PROGRAM FB_Window
VAR
END_VAR
VAR_INPUT
	dataAxis: typeDataAxis;
	optionA:typeVectorOptions;
	optionB:typeVectorOptions;
//	optionC:typeVectorOptions;
//	optionD:typeVectorOptions;
END_VAR

(*
	
	^
	value
	|
	|							C
	|			1_______________________________4
	|			|								|
	|			|								|
	|			|								|
	|			|								|
	|			|								|  
	|		A	|								|  B
	|			|								|
	|			|								|
	|			|								|
	|-----------|----------------line 			|
	|			|_______________________________|
	|			2								3
	|							D
	|							
	|							
	----------------------------------------------------------------time->
	1	2	3	4	5	6	7	8	9 	10 	11	12	13	14	15	16	17 etc
	
	Each side of a box has a entry point, check which vector the data
	passes into


*)


//loop around [4]ness for entire array of data
IF dataAxis.grabTime[4] = optionA.point2.PointXTime THEN //A2 //add in tolerance?
		//evaulate A2
		IF dataAxis.grabData[4] < optionA.point1 OR dataAxis.grabData[4] > optionA.point2 THEN
			//was true
			ELSE
			//was false
		END_IF
END_IF

IF dataAxis.grabTime[4] = optionA.point1.PointXTime THEN //A1 //add in tolerance?
		//evaulate A1
END_IF
///////////////////////////////////////////////////////////////////////////////////

END_PROGRAM

(* stored: Version 1.1.0.1, ProductVersion 3.1.4024.11
   POU FB_Window: Id {4cf7a1dd-4be4-0676-17d1-6d8992ea43f1}, SpecialFunc None *)
